FUNCTION_BLOCK PUBLIC PAESafetyRelay EXTENDS PAESensorDigital
VAR_INPUT
END_VAR
VAR_OUTPUT
END_VAR
VAR
END_VAR

END_FUNCTION_BLOCK

(* stored: Version 1.1.0.1, ProductVersion 3.1.4020.6
   POU PAESafetyRelay: Id {28ccde57-1fca-4b58-9730-ab32d006c2a5}, SpecialFunc None *)
